# EPICS StreamDevice protocol: TM612.proto
##################################################
# General Settings
##################################################

Terminator = CR LF;
ReplyTimeout = 1000;
locktimeout = 5000;
readtimeout  = 1000;
extrainput   = Ignore;

###################################################
# Get functions
###################################################

getTempA {
   out "INPUT A:TEMP?";
   in "%f";
}

getTempB {
   out "INPUT B:TEMP?";
   in "%f";
}

getFieldorCurrent {
   out "IMAG?";
   in "%f";
}

getVoltage {
   out "VMAG?";
   in "%f";
}

getOutputCurrent {
   out "IOUT?";
   in "%f";
}

getOutputVoltage {
   out "VOUT?";
   in "%f";
}

getError {
   out "ERROR?";
   in "%b";
}

getSTB {
   out "*STB?";
   in "%i";
}

getSweep {
   out "SWEEP?";
   in "%s";
}

getMode {
   out "MODE?";
   in "%s";
}

getPSwitch {
   out "PSHTR?";
   in "%i";
}

getRange0 {
   out "RANGE? 0";
   in "%f";
}

getRange1 {
   out "RANGE? 1";
   in "%f";
}

getRange2 {
   out "RANGE? 2";
   in "%f";
}

getRange3 {
   out "RANGE? 3";
   in "%f";
}

getRange4 {
   out "RANGE? 4";
   in "%f";
}

getUnits {
   out "UNITS?";
   in "%s";
}

getLowerSweepLimit {
   out "LLIM?";
   in "%f";
}

getRate0 {
   out "RATE? 0";
   in "%f";
}

getRate1 {
   out "RATE? 1";
   in "%f";
}

getRate2 {
   out "RATE? 2";
   in "%f";
}

getRate3 {
   out "RATE? 3";
   in "%f";
}

getRate4 {
   out "RATE? 4";
   in "%f";
}

getRate5 {
   out "RATE? 5";
   in "%f";
}

getUpperSweepLimit{
   out "ULIM?";
   in "%f";
}

getVLimit {
   out "VLIM?";
   in "%f";
}

######################################################
#Set Functions
######################################################
setPersHeater {
  out "PSHTR %{Off|On}" ;
#  in  "%s";
}
#Could add SWEEP UP FAST but for protection not added
setSweep {
  out "SWEEP %{UP|DOWN|PAUSE|ZERO} SLOW" ;
#  in  "";
}

setUpperSweepLimit {
  out "ULIM %.3f" ;
#  in  "%f";
}

setLowerSweepLimit {
  out "LLIM %.3f" ;
#  in  "%f";
}

setVoltageLimit {
  out "VLIM %.2f" ;
#  in  "%f";
}

setLocal{
  out "RWLOCK" ;
#  in  "%f";
}

setUnits{
 out "UNITS %{G|A}" ;
#  in  "%f";
}
